{attribute 'GeneratedUsingTerminal: EP6002-0002-0016'}
{attribute addProperty BoxType "EP6002-0002-0016"}
{attribute addProperty Id "COM_Inputs_Channel_1AT %I*COM_Inputs_Channel_C252EAC224COM_Inputs_Channel_2AT %I*COM_Inputs_Channel_C252EAC224COM_Outputs_Channel_1AT %Q*COM_Outputs_Channel_B336F4EE24COM_Outputs_Channel_2AT %Q*COM_Outputs_Channel_B336F4EE24WcStateAT %I*WcState_9091E0EB2InfoDataAT %I*InfoData_32EB74EA10"}
{attribute addProperty CRC "644067502"}
{attribute addProperty Size "108"}
TYPE EP6002_2663B0AE :
STRUCT
	{attribute addProperty Name "COM_Inputs_Channel_1"}
	COM_Inputs_Channel_1 : COM_Inputs_Channel_C252EAC2;
	{attribute addProperty Name "COM_Inputs_Channel_2"}
	COM_Inputs_Channel_2 : COM_Inputs_Channel_C252EAC2;
	{attribute addProperty Name "COM_Outputs_Channel_1"}
	COM_Outputs_Channel_1 : COM_Outputs_Channel_B336F4EE;
	{attribute addProperty Name "COM_Outputs_Channel_2"}
	COM_Outputs_Channel_2 : COM_Outputs_Channel_B336F4EE;
	{attribute addProperty Name "WcState"}
	WcState : WcState_9091E0EB;
	{attribute addProperty Name "InfoData"}
	InfoData : InfoData_32EB74EA;
END_STRUCT
END_TYPE

(* stored: Version 1.2.0.0, ProductVersion 3.1.4024.9
   DUT EP6002_2663B0AE: Id {7d8bbaf6-d270-4185-9c0c-c19bbba149b6} *)
